// CALCULATE THE CURRENT OUTFLOW [m3/s]

FUNCTION GetOutFlow : REAL

VAR
	// Module A []
	a : REAL := 14 * EXPT(10,-6);
	
	// Module B []
	b : REAL := SQRT(2 * const.grav * High.now);
	
	// Combine MA and MB []
	coef : REAL := a * b;
	
	
	// Outlet valve value [0-100%]
	valve : REAL := userin.out_percent;

	// Flow in and out [m3/s]
	in  : REAL := flow.in;
	out : REAL;
	
	// Auto hold is enabled?
	match : BOOL := userin.IO_match;

END_VAR

// Calculate output
out := coef * valve;

IF out < 0 THEN
	out := 0;
END_IF

// Return flow value
GetOutFlow := out;
flow.out := out;

// If running IO matching
// Try to find a valve setting to equate in and out
IF match THEN
	userin.out_percent := valve + (in-out)*1000;
END_IF

END_FUNCTION

(* stored: Version 1.1.0.1, ProductVersion 3.1.4024.12
   POU GetOutFlow: Id {9eb8b10c-54cd-4142-b2a4-1aa0751dd7b0}, SpecialFunc None *)
